SUBAPPLICATION Uebung_217 (* Standard IEC 61131-3 FB_CTD_LINT (Rückwärtszähler, LINT) *)
  (* Standard: 61131-3; Description: Copyright (c) 2026 Meisterschulen am Ostbahnhof This program and the accompanying materials are made available under the terms of the Eclipse Public License 2.0 which is available at https://www.eclipse.org/legal/epl-2.0/ SPDX-License-Identifier: EPL-2.0 *)
  (* Version 1.0, 2026-04-20, Franz Höpfinger, Meisterschulen am Ostbahnhof, initial API and implementation (IEC 61131-3 version) *)
  PACKAGE Uebungen;
  IMPORT logiBUS::io::DI::logiBUS_DI::Input_I1;
  IMPORT logiBUS::io::DI::logiBUS_DI::Input_I2;
  IMPORT logiBUS::io::DQ::logiBUS_DO::Output_Q1;
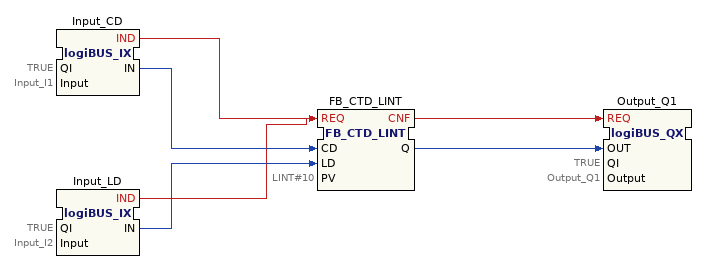
  FBS
    FB_CTD_LINT : iec61131::counters::FB_CTD_LINT(PV := LINT#10);
    Input_CD : logiBUS::io::DI::logiBUS_IX(QI := TRUE, Input := Input_I1);
    Input_LD : logiBUS::io::DI::logiBUS_IX(QI := TRUE, Input := Input_I2);
    Output_Q1 : logiBUS::io::DQ::logiBUS_QX(QI := TRUE, Output := Output_Q1);
  END_FBS
  EVENT_CONNECTIONS
    Input_CD.IND TO FB_CTD_LINT.REQ;
    Input_LD.IND TO FB_CTD_LINT.REQ;
    FB_CTD_LINT.CNF TO Output_Q1.REQ;
  END_CONNECTIONS
  DATA_CONNECTIONS
    Input_CD.IN TO FB_CTD_LINT.CD;
    Input_LD.IN TO FB_CTD_LINT.LD;
    FB_CTD_LINT.Q TO Output_Q1.OUT;
  END_CONNECTIONS
END_SUBAPPLICATION
